Universal Robots PolyScope program: prueba.urp

Program prueba (installation=default directory=/home/ur/ursim-current/programs createdIn=5.7.0.90932 lastSavedIn=5.7.0.90932 robotSerialNumber=20195599999)
Calibrated DH parameters: a=[0, -0.425, -0.3922, 0, 0, 0]; d=[0.1625, 0, 0, 0.1333, 0.0997, 0.0996]; alpha=[1.570796, 0, 0, 1.570796, -1.570796, 0]; deltaTheta=[0, 0, 0, 0, 0, 0]
Robot Program (runOnlyOnce=true)
  Script file /home/ur/ursim-current/programs/prueba.script
    | #info usuario
    | popup("iniciando programa",title="Titulo",warning=False,blocking=True)
    | textmsg("Iniciando programa")
    | 
    | # Preparar instalación
    | set_gravity([0,0,9.8])
    | set_tcp(p[0,0,0.150,0,0,1.57])
    | set_payload_mass(1.5)
    | pi=acos(-1.0)
    | 
    | # Movimiento inicial
    | safe_pose=[0,-0.78,-1.57,-2.15,1.57,0]
    | 
    | movej(safe_pose,pi,1)
    | 
    | # movimientos
    | 
    | pose_1=p[0.5,0,0.25,0,pi,0]
    | pose_2=p[0.5,0,0,0,pi,0]
    | 
    | movej(pose_1,1.5,1)
    | movel(pose_2,1.5,1)
